PROGRAM MAIN
VAR
	a:INT
	b:INT
	c:INT
END_VAR

c:=a+b;

END_PROGRAM

(* stored: Version 1.1.0.1, ProductVersion 3.1.4024.3
   POU MAIN: Id {2313c682-d879-48a2-96b0-58809e4ce1e8}, SpecialFunc None *)
